FUNCTION_BLOCK FB_System_MVHW_300
VAR_INPUT
	Freigabe_auto			: BOOL;
	Freigabe_Deakt_auto		: BOOL:= TRUE;
	Betrieb_Anford_auto		: BOOL;
END_VAR
VAR_OUTPUT
	{attribute 'OPC.UA.DA' := '1'}Steuerung				: ST_System_MVHW_Steuerung;		
	{attribute 'OPC.UA.DA' := '1'}Stellwert				: ST_System_MVHW_Stellwert;		
	{attribute 'OPC.UA.DA' := '1'}Zustand					: ST_System_MVHW_Zustand;	
	{attribute 'OPC.UA.DA' := '1'}Parameter				: ST_System_MVHW_Parameter;		
END_VAR
VAR
	Pumpe_300							: FB_PU;
	Stellventil_300						: FB_SV;
	Maschinenversorgung_JAVA_300		: FB_MV_JAVA;

	Zustandscheck			: FB_System_MVHW_Zustandscheck;
	Logik					: FB_System_MVHW_Logik;
	Ablaufsteuerung			: FB_System_MVHW_Ablaufsteuerung;
END_VAR
VAR // added by the converter: edge detectors and wires of the graphical bodies
    _w1, _w4, _w5 : ANY;
    _w2, _w3 : BOOL;
END_VAR

Steuerung.Freigabe.auto := Freigabe_auto;
Steuerung.Freigabe_Deakt.auto := Freigabe_Deakt_auto;
Steuerung.Betrieb_Anford.auto := Betrieb_Anford_auto;
Parameter := Initialisierung.System_MVHW_Parameter;
Zustandscheck(
    Stellventil_Zustand := Stellventil_300.Zustand,
    Pumpe_Zustand := Pumpe_300.Zustand,
    MV_JAVA_Zustand := Maschinenversorgung_JAVA_300.Zustand,
    MV_JAVA_Parameter := Maschinenversorgung_JAVA_300.Parameter,
    Steuerung := Steuerung,
    Zustand := Zustand); // FB_System_MVHW_Zustandscheck
Logik(Parameter := Parameter, Steuerung := Steuerung, Zustand := Zustand); // FB_System_MVHW_Logik
Ablaufsteuerung(
    Zustand_Stellventil := Stellventil_300.Zustand,
    Zustand_Pumpe := Pumpe_300.Zustand,
    Zustand := Zustand,
    Stellwert := Stellwert,
    Steuerung := Steuerung); // FB_System_MVHW_Ablaufsteuerung
_w1 := Maschinenversorgung_JAVA_300.Zustand.Beheizung_Aktiv OR Zustand.Freigabe;
Stellventil_300(
    Freigabe_auto := _w1,
    Freigabe_Deakt_auto := NOT (_w1 AND NOT _w2),
    Stellung_Anford_auto := Stellwert.Anford_Stellventil,
    Quittierung := Zustand.Quittierung,
    Parameter_init := Initialisierung.Stellventil_300_Parameter); // FB_SV
_w2 := Zustand.Freigabe_Deakt AND NOT Pumpe_300.Zustand.Betrieb;
_w4 := Maschinenversorgung_JAVA_300.Zustand.Beheizung_Aktiv OR _w3;
_w5 := _w3 AND NOT Zustand.Freigabe_Deakt;
_w3 := Zustand.Freigabe AND Stellventil_300.Zustand.Stellung;
Pumpe_300(
    Freigabe_auto := _w4,
    Freigabe_Deakt_auto := NOT _w5,
    Betrieb_Anford_auto := Stellwert.Anford_Pumpe,
    Regelung_Modus_auto := E_PU_Regelung_Modus_dT,
    Regelung_Sollw_auto := 5,
    Quittierung := Zustand.Quittierung,
    Parameter_init := Initialisierung.Pumpe_300_Parameter); // FB_PU
Maschinenversorgung_JAVA_300(Parameter_init := Initialisierung.Anlage_MVHW_Parameter); // FB_MV_JAVA

END_FUNCTION_BLOCK

(* stored: Version 1.1.0.1, ProductVersion 3.1.4024.9
   POU FB_System_MVHW_300: Id {0df92d51-21f9-46c2-8bf8-c85b005e8de2}, SpecialFunc None *)
